// TIA Portal V18 export
// export: Created 2025-12-01T17:51:12.1411829Z, ExportSetting None, DisplayName Totally Integrated Automation Portal, DisplayVersion V18 Update 5, DisplayName TIA Portal Openness, DisplayVersion V18 Update 5, DisplayName TIA Portal Teamcenter Gateway, DisplayVersion V18, DisplayName TIA Portal Version Control Interface, DisplayVersion V18, DisplayName STEP 7 Professional, DisplayVersion V18 Update 5, DisplayName STEP 7 Safety, DisplayVersion V18, DisplayName WinCC Professional, DisplayVersion V18 Update 5
DATA_BLOCK "IAI_Position_DB"   // DB2210
// stored: AutoNumber false, InstanceOfName IAI_Position, InstanceOfType FB
"IAI_Position"
   // VAR
   //    Servo5 { S7_SetPoint := 'True'} : "SevroStart&PosCheck_IAI";
   //    Servo6 { S7_SetPoint := 'True'} : "SevroStart&PosCheck_IAI";
   //    Servo7 { S7_SetPoint := 'True'} : "SevroStart&PosCheck_IAI";
   // END_VAR
BEGIN
END_DATA_BLOCK
